# B&R Automation Studio project IntelliRack
Automation Studio 3.0.80.25

## Logical view

Binary libraries used (declarations not repeated): Visapi, runtime, operator, DataObj, Convert, asstring, AsMath, AsIOAcc

### Global.typ
```iecst
TYPE
	color : STRUCT
		fore	:USINT;
		back	:USINT;
	END_STRUCT;
			ctrlPassword : STRUCT
		levelDatapoint	:UINT;
	END_STRUCT;
			ctrlStatusDatapoint : STRUCT
		ctrlHide	:BOOL;
		ctrlLock	:BOOL;
		ctrlFocus	:BOOL;
		ctrlTouchpad	:BOOL;
		statTouchpad	:BOOL;
		statPressLocked	:BOOL;
		statFocus	:BOOL;
		statEdit	:BOOL;
	END_STRUCT;
			greiferParameter : STRUCT
		pulseWidth	:INT;
		periodDuration	:UINT;
		pulseWidthCurrent	:INT;
		periodDurationCurrent	:UINT;
	END_STRUCT;
			tInp : STRUCT
		overloadDC	:BOOL;
		liftHighLim	:BOOL;
		liftLowLim	:BOOL;
		liftPositionClock	:BOOL;
		wireCoilStrtRight	:BOOL;
		wireCoilStrtLeft	:BOOL;
		wireCoilStpRight	:BOOL;
		wireCoilStpLeft	:BOOL;
		wireCoilEmptyRight	:BOOL;
		wireCoilEmptyLeft	:BOOL;
		sthInPos	:BOOL;
		porStopPos	:BOOL;
		clewJam	:BOOL;
		airPresureOk	:BOOL;
		oilLevelLow	:BOOL;
		oilPresureOk	:BOOL;
		zPosStepper	:BOOL;
		supLeftOff	:BOOL;
		supRightOff	:BOOL;
		supLeftOn	:BOOL;
		supRightOn	:BOOL;
		emgCtrl	:BOOL;
		emgBtn	:BOOL;
		strtBtn	:BOOL;
		stpBtn	:BOOL;
		potiClock	:BOOL;
		potiDirection	:BOOL;
		safetySwitch	:BOOL;
		benderNbr1	:BOOL;
		greaseMainGearOk	:BOOL;
		greaseMainGearErr	:BOOL;
		greaseStepWheelOk	:BOOL;
		greaseStepWheelErr	:BOOL;
	END_STRUCT;
			tStepperControl : STRUCT
		switchOn	:BOOL;
		enbleVoltage	:BOOL;
		quickStop	:BOOL;
		enableOperation	:BOOL;
		faultReset	:BOOL;
		rMotorIdent	:BOOL;
		rResetWarning	:BOOL;
	END_STRUCT;
			tStepperIfIn : STRUCT
		absPosActVal	:DINT;
		status	:UINT;
		inputStatus	:USINT;
	END_STRUCT;
			tStepperIfOut : STRUCT
		absPosSetVal	:DINT;
		control	:UINT;
		mode	:SINT;
	END_STRUCT;
			tStepperStatus : STRUCT
		readyToSwitchOn	:BOOL;
		switchedOn	:BOOL;
		operationEnabled	:BOOL;
		fault	:BOOL;
		voltageEnabled	:BOOL;
		quickStop	:BOOL;
		switchOnDisabeld	:BOOL;
		warning	:BOOL;
		targetReached	:BOOL;
	END_STRUCT;
END_TYPE
```

### Global.var
```iecst
VAR
	Inp	:tInp;
	PeriodDurationPWM01PWM02	:UINT;
	PulseWidthCurrentPWM01	:INT;
	TaskNr	:UINT;
	currentPage	:UINT;
	movePointRef	:ARRAY [0..3] OF BOOL;
	moveStepperNegative	:ARRAY [0..3] OF BOOL;
	moveStepperPositive	:ARRAY [0..3] OF BOOL;
	movesteppos	:DINT;
	rPointReached	:BOOL;
	stStepperControl	:ARRAY [0..3] OF tStepperControl;
	stStepperIfIn	:ARRAY [0..3] OF tStepperIfIn;
	stStepperIfOut	:ARRAY [0..3] OF tStepperIfOut;
	stStepperStatus	:ARRAY [0..3] OF tStepperStatus;
END_VAR
```

### Program Logical/test (IEC, version 1.00.0)

#### testCyclic.ab
```automation-basic
PROGRAM _CYCLIC
(* cyclic program *)

loop	idxDrive	:=	1	to	3	do
	if	(moveToPointRef[idxDrive]=TRUE) or (moveToPointRefAll=TRUE) then
		movePointRef[idxDrive]	:=	1
	else
		movePointRef[idxDrive]	:=	0
	endif
endloop
END_PROGRAM
```

#### test.var
```iecst
VAR
	idxDrive	:DINT;
	moveToPointRef	:ARRAY [0..3] OF BOOL;
	moveToPointRefAll	:BOOL;
END_VAR
```

### Program Logical/sthstep (IEC, version 1.02.0)

#### sthstepCyclic.ab
```automation-basic
PROGRAM _CYCLIC
(* cyclic program *)

; V1.00 	sva		2009-06-17	New
; V1.01
; V1.02		sva		2009-08-14	Handling of restart after emergency stop changed

loop idxDrive:= 1 to 3 do

	speedJog[idxDrive]	:= 20*speedJogOptions[idxDrive]

	gearFactor[idxDrive]				:=  (real(driveStepPerRevolution[idxDrive]) * real(microStepPerDriveStep[idxDrive]) * real(gearZ2[idxDrive]) ) / (real(gearZ1[idxDrive]) * real(gearSlope[idxDrive]))
	referencePositionMicroStep[idxDrive]	:= dint(real(referencePositionMM[idxDrive]) * gearFactor[idxDrive])

	; Get status bits
	; ---------------

	stStepperStatus[idxDrive].readyToSwitchOn		:= bit_tst(stStepperIfIn[idxDrive].status, 0)
	stStepperStatus[idxDrive].switchedOn				:= bit_tst(stStepperIfIn[idxDrive].status, 1)
	stStepperStatus[idxDrive].operationEnabled	:= bit_tst(stStepperIfIn[idxDrive].status, 2)
	stStepperStatus[idxDrive].fault							:= bit_tst(stStepperIfIn[idxDrive].status, 3)
	stStepperStatus[idxDrive].voltageEnabled		:= bit_tst(stStepperIfIn[idxDrive].status, 4)
	stStepperStatus[idxDrive].quickStop					:= bit_tst(stStepperIfIn[idxDrive].status, 5)
	stStepperStatus[idxDrive].switchOnDisabeld	:= bit_tst(stStepperIfIn[idxDrive].status, 6)
	stStepperStatus[idxDrive].warning						:= bit_tst(stStepperIfIn[idxDrive].status, 7)
	stStepperStatus[idxDrive].targetReached			:= bit_tst(stStepperIfIn[idxDrive].status, 10)

	; Drive activated and emergency stopp not pressed
	if (driveActive[idxDrive] = 1) then

		; New referencing
		if (referenceSet[idxDrive] = 255) then
			stStepperControl[idxDrive].enbleVoltage			:= 0
			stStepperControl[idxDrive].quickStop				:= 0
			stStepperControl[idxDrive].switchOn					:= 0
			stStepperControl[idxDrive].enableOperation	:= 0
			referenceSet[idxDrive]											:= 0
			sStepper[idxDrive]													:= sTEP_INIT
		endif

		; State machine stepper
		; ---------------------

		; Emergency stop pressed
;		if (Inp.emgCtrl = 1) then
;			sStepper[idxDrive]	:= sTEP_EMERGENCY_STOP
;		endif

		; Stepper error
		if (stStepperStatus[idxDrive].fault = 1) then
			sStepper[idxDrive]	:= sTEP_ERROR
		endif

		case sStepper[idxDrive] of

			action 0:	; Init step

				stStepperControl[idxDrive].enbleVoltage	:= 1
				stStepperControl[idxDrive].quickStop		:= 1

				if (stStepperStatus[idxDrive].readyToSwitchOn = 1) then

					stStepperControl[idxDrive].switchOn	:= 1

					if (stStepperStatus[idxDrive].switchedOn = 1) then

						stStepperControl[idxDrive].enableOperation	:= 1

						; Drive reference not set
						if (referenceSet[idxDrive] = 0) and (referenceUsed[idxDrive]=TRUE) then
							sStepper[idxDrive]						:= sTEP_MOVE_REFERENCE
							stStepperIfOut[idxDrive].mode	:= modeReference[idxDrive]
						endif

						; Drive reference is set
						if (referenceSet[idxDrive] = 1) or (referenceUsed[idxDrive]=FALSE) then
							sStepper[idxDrive]						:= sTEP_WAIT
							stStepperIfOut[idxDrive].mode	:= mODE_MOVE_POSITION
						endif
					endif
				endif

			endaction

			action 12:	; sTEP_MOVE_REFERENCE

				; Refenece sensor reached
				if (stStepperStatus[idxDrive].targetReached = 1) then
					sStepper[idxDrive]										:= sTEP_SET_REFERENCE_POSITION
					stStepperIfOut[idxDrive].absPosSetVal	:= referencePositionMicroStep[idxDrive]
				endif

			endaction

			action 14:	; sTEP_SET_REFERENCE_POSITION

				; Reference position set
				if (stStepperStatus[idxDrive].targetReached = 1) then
					stStepperIfOut[idxDrive].mode	:= mODE_SET_POSITION
					sStepper[idxDrive]						:= sTEP_WAIT
					referenceSet[idxDrive]				:= 1
					firstMovement[idxDrive]				:= 1
					timerStartUp[idxDrive]				:= 0
				endif

			endaction

			action 20:	; sTEP_WAIT

				if (timerStartUp[idxDrive] <= 200) then
					inc(timerStartUp[idxDrive])
				endif

				; Automatic moving
(*				if (movePos[idxDrive] = 1) then
					; Drive stopped
					if (stStepperStatus[idxDrive].targetReached = 1) and (timerStartUp[idxDrive] > 200) then
						if (oldSetPosition[idxDrive] <> setPosition[idxDrive]) or (firstMovement[idxDrive] = 1) then
							firstMovement[idxDrive]		:= 0
							oldSetPosition[idxDrive]	:= setPosition[idxDrive]
							stStepperIfOut[idxDrive].absPosSetVal	:= (dint(   ((setPosition[idxDrive] / 2)+ mOVING_OFFSET) * gearFactor[idxDrive]))
							stStepperIfOut[idxDrive].mode					:= mODE_MOVE_POSITION
							sStepper[idxDrive]										:= sTEP_MOVE_APPROX_POS
							timer[idxDrive]												:= 0
						endif
					endif
				else
*)
					if (moveStepperPositive[idxDrive]=TRUE) and not (endPointPositive[idxDrive] < stStepperIfIn[idxDrive].absPosActVal) then
						stStepperIfOut[idxDrive].absPosSetVal	:= speedJog[idxDrive]
						stStepperIfOut[idxDrive].mode					:= mODE_MOVE_JOG
						sStepper[idxDrive]										:= sTEP_MOVE_JOG
					else if (moveStepperNegative[idxDrive]=TRUE) and not (endPointNegative[idxDrive] > stStepperIfIn[idxDrive].absPosActVal) then
						stStepperIfOut[idxDrive].absPosSetVal	:= -speedJog[idxDrive]
						stStepperIfOut[idxDrive].mode					:= mODE_MOVE_JOG
						sStepper[idxDrive]										:= sTEP_MOVE_JOG
					else if	(setPointZero[idxDrive]=TRUE)	then
						zeroPoint[idxDrive]										:= stStepperIfIn[idxDrive].absPosActVal
						refPointMove[idxDrive]								:= DINT(((REAL(refPoint[idxDrive])+REAL(zeroPoint[idxDrive]))/1024)*200*256)
					else if (movePointRef[idxDrive]=TRUE) then
						stStepperIfOut[idxDrive].absPosSetVal	:= refPointMove[idxDrive]
						stStepperIfOut[idxDrive].mode					:= mODE_MOVE_POSITION
						sStepper[idxDrive]										:= sTEP_MOVE_APPROX_POS
					else if (currentPage = 0) then
						stStepperIfOut[1].absPosSetVal				:= movesteppos
						stStepperIfOut[1].mode								:= mODE_MOVE_POSITION
						sStepper[1]														:= 30
					endif
;				endif

				; Switch on disabled
				if (stStepperStatus[idxDrive].switchOnDisabeld = 1) then
					stStepperControl[idxDrive].switchOn	:= 0
					sStepper[idxDrive]									:= sTEP_SHUTDOWN
				endif

			endaction

			action 21: ;sTEP_MOVE_APPROX_POS

				; Moved to set position + offset
				if (stStepperStatus[idxDrive].targetReached = 1) then
					stStepperIfOut[idxDrive].absPosSetVal	:= refPointMove[idxDrive]
					stStepperIfOut[idxDrive].mode					:= mODE_MOVE_POSITION
					sStepper[idxDrive]										:= sTEP_MOVE_FINE_POS
				endif

				; Switch on disabled
				if (stStepperStatus[idxDrive].switchOnDisabeld = 1) then
					stStepperControl[idxDrive].switchOn	:= 0
					sStepper[idxDrive]									:= sTEP_SHUTDOWN
				endif

			endaction

			action 22:		; sTEP_MOVE_FINE_POS

				; Moved to set position
				if (stStepperStatus[idxDrive].targetReached = 1) then
					sStepper[idxDrive]	:= sTEP_WAIT
				endif

				; Switch on disabled
				if (stStepperStatus[idxDrive].switchOnDisabeld=1) then
					stStepperControl[idxDrive].switchOn	:= 0
					sStepper[idxDrive]									:= sTEP_SHUTDOWN
				endif

			endaction

			action 23: ; sTEP_MOVE_JOG

			endPointNegative[1]	:= zeroPoint[1] - 2200
			endPointNegative[2]	:= zeroPoint[2] - 3800
			endPointNegative[3]	:= zeroPoint[3] - 1280 - 59

			endPointPositive[1]	:= zeroPoint[1] + 2304
			endPointPositive[2]	:= zeroPoint[2]
			endPointPositive[3]	:= zeroPoint[3] - 59

				; Switch on disabled
				if (stStepperStatus[idxDrive].switchOnDisabeld = 1) then
					stStepperControl[idxDrive].switchOn	:= 0
					sStepper[idxDrive]									:= sTEP_SHUTDOWN
				endif

				if ((moveStepperPositive[idxDrive]=FALSE) or (endPointPositive[idxDrive] < stStepperIfIn[idxDrive].absPosActVal)) and ((moveStepperNegative[idxDrive]=FALSE) or (endPointNegative[idxDrive] > stStepperIfIn[idxDrive].absPosActVal)) then
					stStepperIfOut[idxDrive].absPosSetVal	:= 0
					sStepper[idxDrive]										:= sTEP_SHUTDOWN
				endif

			endaction

			action 24:	;sTEP_MOVE_REF

				; Switch on disabled
				if (stStepperStatus[idxDrive].switchOnDisabeld = 1) then
					stStepperControl[idxDrive].switchOn	:= 0
					sStepper[idxDrive]									:= sTEP_SHUTDOWN
				endif

				if (movePointRef[idxDrive]=FALSE) then
					sStepper[idxDrive]	:= sTEP_WAIT
				endif

			endaction

			action 25:	; sTEP_SHUTDOWN

				; Switch on enabled
				if (stStepperStatus[idxDrive].switchOnDisabeld = 0) then
					stStepperControl[idxDrive].switchOn	:= 1
					sStepper[idxDrive]									:= sTEP_WAIT
				endif

			endaction

			action 30:
				if (stStepperStatus[idxDrive].switchOnDisabeld = 1) then
					stStepperControl[idxDrive].switchOn	:= 0
					sStepper[idxDrive]									:= sTEP_SHUTDOWN
				endif

				if 1 = 1 then
					sStepper[idxDrive]	:= sTEP_WAIT
				endif

			endaction

			action 250:	; Emergency stopp

				stStepperControl[idxDrive].enableOperation	:= 0

				; Emergency stop released
				if (Inp.emgCtrl=0) then
					stStepperControl[idxDrive].enbleVoltage	:= 1
					stStepperControl[idxDrive].quickStop		:= 1
					sStepper[idxDrive]											:= sTEP_INIT
				endif

			endaction

			action 255:	; Error step

				stStepperControl[idxDrive].enbleVoltage			:= 0
				stStepperControl[idxDrive].quickStop				:= 0
				stStepperControl[idxDrive].switchOn					:= 0
				stStepperControl[idxDrive].enableOperation	:= 0
				stStepperControl[idxDrive].faultReset				:= 1

				if (stStepperStatus[idxDrive].fault=0) then
					stStepperControl[idxDrive].enbleVoltage	:= 1
					stStepperControl[idxDrive].quickStop		:= 1
					sStepper[idxDrive]											:= sTEP_INIT
				endif

			endaction

		endcase

	; Not active
	else

		stStepperControl[idxDrive].enbleVoltage			:= 0
		stStepperControl[idxDrive].quickStop				:= 0
		stStepperControl[idxDrive].switchOn					:= 0
		stStepperControl[idxDrive].enableOperation	:= 0
		oldWireLengthMM[idxDrive]										:= 0
		sStepper[idxDrive]													:= sTEP_INIT
		referenceSet[idxDrive]											:= 0

	endif

	; Set control word
	; ----------------

	if (stStepperControl[idxDrive].switchOn=1) then
		stStepperIfOut[idxDrive].control	:= bit_set(stStepperIfOut[idxDrive].control, 0)
	else
		stStepperIfOut[idxDrive].control	:= bit_clr(stStepperIfOut[idxDrive].control, 0)
	endif

	if (stStepperControl[idxDrive].enbleVoltage=1) then
		stStepperIfOut[idxDrive].control	:= bit_set(stStepperIfOut[idxDrive].control, 1)
	else
		stStepperIfOut[idxDrive].control	:= bit_clr(stStepperIfOut[idxDrive].control, 1)
	endif

	if (stStepperControl[idxDrive].quickStop=1) then
		stStepperIfOut[idxDrive].control	:= bit_set(stStepperIfOut[idxDrive].control, 2)
	else
		stStepperIfOut[idxDrive].control	:= bit_clr(stStepperIfOut[idxDrive].control, 2)
	endif

	if (stStepperControl[idxDrive].enableOperation=1) then
		stStepperIfOut[idxDrive].control	:= bit_set(stStepperIfOut[idxDrive].control, 3)
	else
		stStepperIfOut[idxDrive].control	:= bit_clr(stStepperIfOut[idxDrive].control, 3)
	endif

	if (stStepperControl[idxDrive].faultReset=1) then
		stStepperControl[idxDrive].faultReset	:= 0
		stStepperIfOut[idxDrive].control				:= bit_set(stStepperIfOut[idxDrive].control, 7)
	else
		stStepperIfOut[idxDrive].control	:= bit_clr(stStepperIfOut[idxDrive].control, 7)
	endif

	if (stStepperControl[idxDrive].rMotorIdent=1) then
		stStepperControl[idxDrive].rMotorIdent	:= 0
		stStepperIfOut[idxDrive].control					:= bit_set(stStepperIfOut[idxDrive].control, 11)
	else
		stStepperIfOut[idxDrive].control	:= bit_clr(stStepperIfOut[idxDrive].control, 11)
	endif

	if (stStepperControl[idxDrive].rResetWarning=1) then
		stStepperControl[idxDrive].rResetWarning	:= 0
		stStepperIfOut[idxDrive].control						:= bit_set(stStepperIfOut[idxDrive].control, 12)
	else
		stStepperIfOut[idxDrive].control	:= bit_clr(stStepperIfOut[idxDrive].control, 12)
	endif

	if (stStepperControl[idxDrive].enableOperation=1) then
		stStepperIfOut[idxDrive].control	:= bit_set(stStepperIfOut[idxDrive].control, 14)
	else
		stStepperIfOut[idxDrive].control	:= bit_clr(stStepperIfOut[idxDrive].control, 14)
	endif

	; MMI aufgestartet d.h. alle Daten aktuell
;	if (dMMI.picture.idxActPic<>0) then
		driveActive[idxDrive]	:= 1
;	endif

endloop
END_PROGRAM
```

#### sthstepInit.ab
```automation-basic
PROGRAM _INIT
(* init program *)
inc(TaskNr)

speedJogOptions[1]	:=	25
speedJogOptions[2]	:=	15
speedJogOptions[3]	:=	10

refPoint[1]	:=	1152
refPoint[2]	:=	-1733
refPoint[3]	:=	-59

zeroPoint[2]	:=	4000

loop idxDrive:= 1 to 3 do

	referenceUsed[idxDrive]	:= FALSE

	sStepper[idxDrive]			:= sTEP_INIT
	referenceSet[idxDrive]	:= 0
	driveActive[idxDrive]		:= 0					; Nicht aktivieren bis alle Daten vorhanden sind
	movePos[idxDrive]				:= 0					; Automatisches Fahren deaktivieren
	modeReference[idxDrive]	:= -128

	; Init control word
	; -----------------

	stStepperControl[idxDrive].switchOn					:= 0
	stStepperControl[idxDrive].enbleVoltage			:= 1
	stStepperControl[idxDrive].quickStop				:= 1
	stStepperControl[idxDrive].enableOperation	:= 0
	stStepperControl[idxDrive].faultReset				:= 0
	stStepperControl[idxDrive].rMotorIdent			:= 0
	stStepperControl[idxDrive].rResetWarning		:= 0

	;========================================
	;	Step Umrechnung
	;========================================

	gearZ1[idxDrive]									:= 15				; Getriebe Zähnezahl Antrieb
	gearZ2[idxDrive]									:= 40				; Getriebe Zähnezahl Abtrieb
	gearSlope[idxDrive]								:= 2.0			; Steigung Gewindestange
	driveStepPerRevolution[idxDrive]	:= 200			; Steps per drive turning
	microStepPerDriveStep[idxDrive] 	:= 256			; Microsteps of X20 stepper module

	referencePositionMM[idxDrive]			:= real(initPosition[idxDrive]) / 1000			; Resulting (wire length / 2) at reference position

	gearFactor[idxDrive]									:=  (real(driveStepPerRevolution[idxDrive]) * real(microStepPerDriveStep[idxDrive]) * real(gearZ2[idxDrive]) ) / (real(gearZ1[idxDrive])* real(gearSlope[idxDrive]))
	referencePositionMicroStep[idxDrive]	:= dint(real(referencePositionMM[idxDrive]) * gearFactor[idxDrive])

endloop
END_PROGRAM
```

#### sthstep.var
```iecst
VAR RETAIN
	initPosition	:ARRAY [0..3] OF UINT;
END_VAR

VAR CONSTANT
	sTEP_INIT	:USINT	:=0;
	sTEP_EMERGENCY_STOP	:UINT	:=250;
	sTEP_ERROR	:USINT	:=255;
	sTEP_MOVE_REFERENCE	:USINT	:=12;
	mODE_MOVE_POSITION	:SINT	:=1;
	sTEP_WAIT	:USINT	:=20;
	sTEP_SET_REFERENCE_POSITION	:USINT	:=14;
	sTEP_SHUTDOWN	:UINT	:=25;
	mOVING_OFFSET	:REAL	:=0.5;
	sTEP_MOVE_APPROX_POS	:USINT	:=21;
	sTEP_MOVE_FINE_POS	:USINT	:=22;
	mODE_SET_POSITION	:SINT	:=-122;
	mODE_MOVE_JOG	:SINT	:=2;
	sTEP_MOVE_JOG	:UINT	:=23;
	sTEP_MOVE_REF	:USINT	:=24;
END_VAR

VAR
	sStepper	:ARRAY [0..3] OF UINT;
	idxDrive	:USINT;
	stStepperStatus	:ARRAY [0..3] OF tStepperStatus;
	stStepperIfIn	:ARRAY [0..3] OF tStepperIfIn;
	stStepperControl	:ARRAY [0..3] OF tStepperControl;
	wireLengthPositionMM	:ARRAY [0..3] OF REAL;
	referenceSet	:ARRAY [0..3] OF USINT;
	modeReference	:ARRAY [0..3] OF SINT;
	timerStartUp	:ARRAY [0..3] OF UDINT;
	gearZ1	:ARRAY [0..3] OF UDINT;
	gearZ2	:ARRAY [0..3] OF UDINT;
	gearSlope	:ARRAY [0..3] OF REAL;
	microStepPerDriveStep	:ARRAY [0..3] OF UINT;
	driveStepPerRevolution	:ARRAY [0..3] OF UDINT;
	gearFactor	:ARRAY [0..3] OF REAL;
	referencePositionMM	:ARRAY [0..3] OF REAL;
	pMMI	:UDINT;
	gPvXGetAdr	:UINT;
	size	:UINT;
	firstMovement	:ARRAY [0..3] OF USINT;
	stStepperIfOut	:ARRAY [0..3] OF tStepperIfOut;
	wireLengthMM	:ARRAY [0..3] OF REAL;
	oldWireLengthMM	:ARRAY [0..3] OF REAL;
	timer	:ARRAY [0..3] OF INT;
	referencePositionMicroStep	:ARRAY [0..3] OF DINT;
	movePos	:ARRAY [0..3] OF USINT;
	wireLengthOffsetMM	:ARRAY [0..3] OF REAL;
	driveActive	:ARRAY [0..3] OF USINT;
	speedJogOptions	:ARRAY [0..3] OF DINT;
	referenceUsed	:ARRAY [0..3] OF BOOL;
	setPosition	:ARRAY [0..3] OF REAL;
	oldSetPosition	:ARRAY [0..3] OF REAL;
	moveStepperPositive	:ARRAY [0..3] OF BOOL;
	speedJog	:ARRAY [0..3] OF DINT;
	moveStepperNegative	:ARRAY [0..3] OF BOOL;
	moveStepperReference	:ARRAY [0..3] OF BOOL;
	refPoint	:ARRAY [0..3] OF DINT;
	setPointZero	:ARRAY [0..3] OF BOOL;
	zeroPoint	:ARRAY [0..3] OF DINT;
	refPointMove	:ARRAY [0..3] OF DINT;
	detail1	:USINT;
	detail2	:USINT;
	detail4	:USINT;
	detail3	:USINT;
	endPointPositive	:ARRAY [0..3] OF DINT;
	endPointNegative	:ARRAY [0..3] OF DINT;
END_VAR
```

### Program Logical/greifer (IEC, version 1.00.0)

#### greiferCyclic.ab
```automation-basic
PROGRAM _CYCLIC
(* cyclic program *)

if (moveGreiferPositive=TRUE) then
	greifer.pulseWidthCurrent			:=	greifer.pulseWidth
	greifer.periodDurationCurrent	:=	greifer.periodDuration
else if (moveGreiferNegative=TRUE) then
	greifer.pulseWidthCurrent			:=	-greifer.pulseWidth
	greifer.periodDurationCurrent	:=	greifer.periodDuration
else
	greifer.pulseWidthCurrent			:=	0
	greifer.periodDurationCurrent	:=	0
endif
END_PROGRAM
```

#### greiferInit.ab
```automation-basic
PROGRAM _INIT
(* init program *)

;Frequenz							us pro Zyklus
greifer.pulseWidth			:=	5000

;Anteil in "Prozent" (UINT) von 1/-1 Signal
greifer.periodDuration	:=	20
END_PROGRAM
```

#### greifer.var
```iecst
VAR
	moveGreiferPositive	:BOOL;
	moveGreiferNegative	:BOOL;
	greifer	:greiferParameter;
END_VAR
```

### Program Logical/ctrlvisu (IEC, version 0.00.0)

#### ctrlvisuCyclic.ab
```automation-basic
PROGRAM _CYCLIC
(* cyclic program *)

if detail1 = 0 then
	detail1focus := 2
else if detail2 = 0 then
	detail1focus := 2
else if detail3 = 0 then
	detail1focus := 2
else if detail4 = 0 then
	detail1focus := 2
else
	detail1focus := 0
	detail2focus := 0
	detail3focus := 0
	detail4focus := 0
endif

if ready <> 1 then
	VC_HANDLE = VA_Setup(1, "visu")

	if	VC_HANDLE <> 0 then
		ready = 1
	endif
endif

loop idx :=	1 to 5 do

	statusDatapoint[idx].statTouchpad			:=	bit_tst(ctrlWord[idx], 12)
	statusDatapoint[idx].statPressLocked	:=	bit_tst(ctrlWord[idx], 13)
	statusDatapoint[idx].statFocus				:=	bit_tst(ctrlWord[idx], 14)
	statusDatapoint[idx].statEdit					:=	bit_tst(ctrlWord[idx], 15)

endloop
if currentPage <> 0 then
	CASE	achsenwahl of
		action 1:
			if statusDatapoint[5].statFocus = 0 then
				statusDatapoint[1].ctrlHide = 1

				achsenwahl :=	2
			endif
		endaction

		action 2:

			if VA_Saccess(1, VC_HANDLE)= 0 then

				VA_GetTouchAction(1, VC_HANDLE, 0, UDINT(ADR(touch2)))

				if (touch2.status = 1) and (touch2.x > 255) and (touch2.x < 385) and (touch2.y > 420) and (detail1 = 1) and (detail2 = 1) and (detail3 = 1) and (detail4 = 1)then
					statusDatapoint[1].ctrlHide = 0

					achsenwahl := 3
				endif

				VA_Srelease(1, VC_HANDLE)
			endif
		endaction

		action 3:

			if ready = 1 then
				if VA_Saccess(1, VC_HANDLE)= 0 then

					VA_GetTouchAction(1, VC_HANDLE, 0, UDINT(ADR(touch2)))

					if touch2.status = 1 then
						if (touch2.x > 255) and (touch2.x < 385) and (touch2.y > 420) then
							idxbmp	:=	0
						else if (touch2.x > 255) and (touch2.x < 385) and (touch2.y > 380) then
							idxbmp	:=	1
						else if (touch2.x > 255) and (touch2.x < 385) and (touch2.y > 340) then
							idxbmp	:=	2
						else if (touch2.x > 255) and (touch2.x < 385) and (touch2.y > 300) then
							idxbmp	:=	3
						else if (touch2.x > 255) and (touch2.x < 385) and (touch2.y > 260) then
							idxbmp	:=	4
						else
							idxbmp	:=	0
						endif
					else if touch2.status = 2 then
						if (touch2.x > 255) and (touch2.x < 385) and (touch2.y > 420) then
							changePage	:=	12
							achsenwahl	:=	1
						else if (touch2.x > 255) and (touch2.x < 385) and (touch2.y > 380) then
							changePage	:=	6
							achsenwahl	:=	1
						else if (touch2.x > 255) and (touch2.x < 385) and (touch2.y > 340) then
							changePage	:=	7
							achsenwahl	:=	1
						else if (touch2.x > 255) and (touch2.x < 385) and (touch2.y > 300) then
							changePage	:=	3
							achsenwahl	:=	1
						else if (touch2.x > 255) and (touch2.x < 385) and (touch2.y > 260) then
							changePage	:=	4
							achsenwahl	:=	1
						endif
					endif

					VA_Srelease(1, VC_HANDLE)

				endif
			endif
		endaction
	endcase
endif

loop idx := 1 to 5 do

	if statusDatapoint[idx].ctrlFocus = 1 then
		ctrlWord[idx]	:=	bit_set(ctrlWord[idx], 3)
	else if statusDatapoint[idx].ctrlFocus = 0 then
		ctrlWord[idx]	:=	bit_clr(ctrlWord[idx], 3)
	endif

	if statusDatapoint[idx].ctrlLock = 1 then
		ctrlWord[idx]	:=	bit_set(ctrlWord[idx], 1)
	else if statusDatapoint[idx].ctrlLock = 0 then
		ctrlWord[idx]	:=	bit_clr(ctrlWord[idx], 1)
	endif

	if statusDatapoint[idx].ctrlHide = 1 then
		ctrlWord[idx]	:=	bit_set(ctrlWord[idx], 0)
	else if statusDatapoint[idx].ctrlHide = 0 then
		ctrlWord[idx]	:=	bit_clr(ctrlWord[idx], 0)
	endif

	if statusDatapoint[idx].ctrlTouchpad = 1 then
		ctrlWord[idx]	:=	bit_set(ctrlWord[idx], 2)
	else if statusDatapoint[idx].ctrlTouchpad = 0 then
		ctrlWord[idx]	:=	bit_clr(ctrlWord[idx], 2)
	endif
endloop

;Damit die Visualisierung da Passwort ausführen kann
password.levelDatapoint
END_PROGRAM
```

#### ctrlvisuInit.ab
```automation-basic
PROGRAM _INIT
(* init program *)

achsenwahl := 1

detail1 := 1
detail2 := 1
detail3 := 1
detail4 := 1

detail1focus := 0
detail2focus := 0
detail3focus := 0
detail4focus := 0
END_PROGRAM
```

#### ctrlvisu.var
```iecst
VAR
	statusDatapoint	:ARRAY [0..5] OF ctrlStatusDatapoint;
	ctrlWord	:ARRAY [0..5] OF UINT;
	lock	:BOOL;
	hide	:BOOL;
	touchpad	:BOOL;
	focus	:BOOL;
	idx	:UINT;
	achsenwahl	:UINT;
	ready	:BOOL;
	VC_HANDLE	:UDINT;
	test	:BOOL;
	touch2	:TouchAction;
	changePage	:UINT;
	idxbmp	:UINT;
	password	:ctrlPassword;
	durchgang1	:BOOL;
	detail4	:UINT;
	detail1	:UINT;
	detail2	:UINT;
	detail3	:UINT;
	detail1focus	:UINT;
	detail2focus	:UINT;
	detail3focus	:UINT;
	detail4focus	:UINT;
END_VAR
```

### Program Logical/stepmove (IEC, version 0.00.0)

#### stepmoveCyclic.ab
```automation-basic
PROGRAM _CYCLIC
(* cyclic program *)

;Wenn die aktuelle Seite die Experimentierseite ist
if currentPage = 0 then

	;Bildschirm bereit zum Bearbeiten
	if ready <> 1 then
		VC_HANDLE = VA_Setup(1, "visu")

		if	VC_HANDLE <> 0 then
			ready = 1
		endif
	endif

	;Wenn Bildschirm bereit zum Bearbeiten
	if ready = 1 then

		;Erster Durchlauf Formen zeichnen
		if test = 0 then
			if VA_Saccess(1, VC_HANDLE)= 0 then

				;Mittelpunkt zeichnen
				VA_Rect(1, VC_HANDLE, 239, 239, 3, 3, fill, color)

				;Aktuelle-Position Form zeichnen
				VA_Rect(1, VC_HANDLE, UINT(position_x), UINT(position_y), width, heigth, fill, color)
				test = 1

				VA_Srelease(1, VC_HANDLE)

			endif
		endif

		;Weitere Durchläufe
		if test = 1 then

			if VA_Saccess(1, VC_HANDLE) = 0 then

				;Welche Taste ist aktuell betätigt
				if fest = 1 then
					bewegen = 0
				else if locker = 1 then
					bewegen = 1
					zeichnen = 1
					VA_Redraw(1, VC_HANDLE)
					VA_Rect(1, VC_HANDLE, 239, 239, 3, 3, fill, color)
					VA_Rect(1, VC_HANDLE, UINT(position_x), UINT(position_y), width, heigth, fill, color)
				endif

				;Abfragen der aktuelle Touch-Position
				VA_GetTouchAction(1, VC_HANDLE, 0, UDINT(adr(touch)))

				;Übergabe der Touch-Position Informationen
				x_position = touch.x
				y_position = touch.y
				touch_status = touch.status

				;Wenn Touchpanel betätigt und bewegen erlaubt
				if touch_status = 1 and bewegen = 1 then

					;Abfrage ob Form gegriffen wurde
					if ((x_position) > position_x) and ((x_position) < (position_x + width)) and ((y_position) > position_y) and ((y_position) < (position_y + heigth)) and (packen_erlaubt = 0) and bewegen = 1 then
						packen_erlaubt = 1
						gepackt_x = x_position - position_x
						gepackt_y = y_position - position_y

						;Überschreiben der Drawbox mit weiss
						VA_Rect(1, VC_HANDLE, 0, 0, 480, 480, 15, 15)

						;Mittelpunkt zeichnen
						VA_Rect(1, VC_HANDLE, 239, 239, 3, 3, fill, color)
					endif

					;Wenn Form gegriffen wurde
					if packen_erlaubt = 1 then

						;Letzte Position der Form löschen
						VA_Rect(1, VC_HANDLE, UINT(position_x), UINT(position_y), width, heigth, 15, 15)

						;Mittelpunkt zeichnen
						VA_Rect(1, VC_HANDLE, 239, 239, 3, 3, fill, color)

						;Berechnen der Form-Position
						x1 = x1 + (x_position - x_position_old)
						y1 = y1 + (y_position - y_position_old)

						position_x = x1 - gepackt_x
						position_y = y1 - gepackt_y

						;Berechnen der Richtung und Schritte für Drehtisch
						x_position_EXP	:=	(EXPT(-240+x_position,2))
						y_position_EXP	:=	(EXPT(-240+y_position,2))
						sqrtergebnis		:=	SQRT(EXPT(-240+x_position,2))/SQRT((y_position_EXP)+(x_position_EXP))

						if (x_position < 240) and (y_position < 240) then
							asdasd					:=	ASIN(sqrtergebnis)
							asd							:=	90
						else if (x_position > 240) and (y_position < 240) then
							asdasd					:=	ACOS(sqrtergebnis)
							asd							:=	0
						else if (x_position > 240) and (y_position > 240) then
							asdasd					:=	ASIN(sqrtergebnis)
							asd							:=	-90
						else if (x_position < 240) and (y_position > 240) then
							asdasd					:=	ACOS(sqrtergebnis)
							asd							:=	-180
						endif

						dasdas 					:= (25600*((360*asdasd/amTWOPI)+asd))/360
						dasdasdasdasda	:=	DINT(dasdas)

						movesteppos			:= 9*dasdasdasdasda

						;Drawbox-Begrenzungen
						if ((x_position - gepackt_x + width) > x_stop) then
							position_x = x_stop - width
						else if ((x_position - gepackt_x) < x_start) then
							position_x = x_start
						endif

						if ((y_position - gepackt_y + heigth) > y_stop) then
							position_y = y_stop - heigth
						else if ((y_position - gepackt_y) < y_start) then
							position_y = y_start
						endif

						;Zeichnen der Form
						VA_Rect(1, VC_HANDLE, UINT(position_x), UINT(position_y), width, heigth, fill, color)

						;Speichern der letztn Position
						x_position_old = x_position
						y_position_old = y_position

					endif

				else
					if packen_erlaubt = 1 then
						packen_erlaubt = 0
					endif
				endif

				VA_Srelease(1, VC_HANDLE)
			endif
		endif
	endif
endif
END_PROGRAM
```

#### stepmoveInit.ab
```automation-basic
PROGRAM _INIT
(* init program *)

test 						:= 0
x1 							:= 400
y1 							:= 235
x_position_old 	:= x1
y_position_old 	:= y1

;Startposition der From
position_x 			:= 400
position_y 			:= 235

;Parameter für Begrenzungen vom Zeichen
x_start 				:= 0
x_stop					:= 480
y_start					:= 0
y_stop					:= 480

;Paramter für Form der aktuellen Position
heigth					:=	20
width						:=	20
fill						:=	0
color						:=	0
END_PROGRAM
```

#### stepmove.var
```iecst
VAR
	test	:BOOL;
	ready	:BOOL;
	VC_HANDLE	:UDINT;
	redesign	:BOOL;
	packen_erlaubt	:BOOL;
	fest	:BOOL;
	width	:UINT;
	heigth	:UINT;
	touch_status	:UDINT;
	dasdas	:REAL;
	y_start	:DINT;
	x_start	:DINT;
	fill	:UINT;
	x_position	:DINT;
	zeichnen	:BOOL;
	locker	:BOOL;
	x_position_old	:DINT;
	position_x	:DINT;
	y_position_old	:DINT;
	position_y	:DINT;
	y_position	:DINT;
	touch	:TouchAction;
	y_stop	:DINT;
	x_stop	:DINT;
	bewegen	:BOOL;
	asdasd	:REAL;
	y1	:DINT;
	x1	:DINT;
	color	:UINT;
	gepackt_x	:DINT;
	gepackt_y	:DINT;
	dasdasdasdasda	:DINT;
	x_position_EXP	:REAL;
	y_position_EXP	:REAL;
	sqrtergebnis	:REAL;
	asd	:REAL;
	das	:DINT;
END_VAR
```

### Program Logical/testvisu (IEC, version 0.00.0)

#### testvisuCyclic.ab
```automation-basic
PROGRAM _CYCLIC
(* cyclic program *)

;loop	idx	:=	1	to	8	do
;	color	access	adr	(idxColor[idx])
;	color.fore	:=	100
;	color.back	:=	0
;endloop

if (ready <> 1) then
	VC_HANDLE = VA_Setup(1, "visu")

	if	VC_HANDLE <> 0 then
		ready := 1
	endif
endif

if (ready = 1) and (first = 0) then
	if VA_Saccess(1, VC_HANDLE)= 0 then

		VA_Redraw(1, VC_HANDLE)

		VA_Rect(1, VC_HANDLE, 0, 400, 640, 80, 100, 100)

		VA_Srelease(1, VC_HANDLE)

		first	:=	1

	endif
endif

if (ready = 1) and (first = 1) then
	if VA_Saccess(1, VC_HANDLE)= 0 then

		VA_GetTouchAction(1, VC_HANDLE, 0, UDINT(ADR(touch2)))

			Aktion	:=	BOOL(touch2.status - 1)
			;if touch2.status = 1 then

			if EDGE(Aktion) then
				VA_Rect(1, VC_HANDLE, 0, 320, 640, 80, 15, 15)
			endif

			VA_Rect(1, VC_HANDLE, (80 * (changed - 1)), 400, 80, 80, 100, 100)

			loop	idx:=	1	to	8 do

				if (touch2.x	< (80 * idx)) and (touch2.x > (80 * (idx - 1))) and (touch2.y > 399) then
					if (touch2.status = 1) and (counter2 <> 2) then
						changed	:=	idx
						VA_Rect(1, VC_HANDLE, (80 * (idx - 1)), 400, 80, 80, 10, 10)
						counter := 0
						inc(counter2)
					else if (touch2.status = 2) and (counter <> 2) then
						VA_Rect(1, VC_HANDLE, 0, 320, 640, 80, 15, 15)
						VA_Rect(1, VC_HANDLE, (80 * (idx - 1)), 320, 80, 80, 10, 10)
						counter2 :=	0
						inc(counter)
					endif
				endif

			endloop
			;endif

		VA_Srelease(1, VC_HANDLE)

	endif
endif
END_PROGRAM
```

#### testvisuInit.ab
```automation-basic
PROGRAM _INIT
(* init program *)

first := 0
END_PROGRAM
```

#### testvisu.var
```iecst
VAR
	idx	:UINT;
	ready	:BOOL;
	VC_HANDLE	:UDINT;
	touch2	:TouchAction;
	changed	:UINT;
	first	:BOOL;
	Aktion	:BOOL;
	counter2	:USINT;
	counter	:USINT;
END_VAR
```

### Program Logical/testvisa (IEC, version 0.00.0)

#### testvisaCyclic.ab
```automation-basic
PROGRAM _CYCLIC
(* cyclic program *)

(* cyclic program *)

if (ready <> 1) then
	VC_HANDLE = VA_Setup(1, "visu")

	if	VC_HANDLE <> 0 then
		ready := 1
		if VA_Saccess(1, VC_HANDLE)= 0 then
			VA_Redraw(1, VC_HANDLE)
			VA_Srelease(1, VC_HANDLE)
		endif
	endif
endif

if (ready = 1) then
	if VA_Saccess(1, VC_HANDLE)= 0 then

		VA_Rect(1, VC_HANDLE, UINT(touch2.x-40), UINT(touch2.y-40), 80, 80, 15, 15)

		VA_GetTouchAction(1, VC_HANDLE, 0, UDINT(ADR(touch2)))

		VA_Rect(1, VC_HANDLE, UINT(touch2.x-40), UINT(touch2.y-40), 80, 80, UINT((touch2.x/6.4) + (touch2.y/4.8)), UINT((touch2.x/6.4) + (touch2.y/4.8)))

		VA_Srelease(1, VC_HANDLE)

	endif
endif
END_PROGRAM
```

#### testvisa.var
```iecst
VAR
	ready	:BOOL;
	VC_HANDLE	:UDINT;
	touch2	:TouchAction;
END_VAR
```

### Program Logical/a_soption (IEC, version 0.00.0)

#### a_soptionCyclic.ab
```automation-basic
PROGRAM _CYCLIC
(* cyclic program *)

AsIOAccWrite(1, UDINT(ADR("SL1.SS1.IF2.ST16.IF1.ST3")), UDINT(ADR("ConfigOutput03a")), valueHaltestrom[1], status)
AsIOAccWrite(1, UDINT(ADR("SL1.SS1.IF2.ST16.IF1.ST3")), UDINT(ADR("ConfigOutput04a")), valueNennstrom[1], status)
AsIOAccWrite(1, UDINT(ADR("SL1.SS1.IF2.ST16.IF1.ST3")), UDINT(ADR("ConfigOutput05a")), valueMaximalstrom[1], status)

AsIOAccWrite(1, UDINT(ADR("SL1.SS1.IF2.ST16.IF1.ST6")), UDINT(ADR("ConfigOutput03")), valueHaltestrom[2], status)
AsIOAccWrite(1, UDINT(ADR("SL1.SS1.IF2.ST16.IF1.ST6")), UDINT(ADR("ConfigOutput04")), valueNennstrom[2], status)
AsIOAccWrite(1, UDINT(ADR("SL1.SS1.IF2.ST16.IF1.ST6")), UDINT(ADR("ConfigOutput05")), valueMaximalstrom[2], status)

AsIOAccWrite(1, UDINT(ADR("SL1.SS1.IF2.ST16.IF1.ST6")), UDINT(ADR("ConfigOutput06")), valueHaltestrom[3], status)
AsIOAccWrite(1, UDINT(ADR("SL1.SS1.IF2.ST16.IF1.ST6")), UDINT(ADR("ConfigOutput07")), valueNennstrom[3], status)
AsIOAccWrite(1, UDINT(ADR("SL1.SS1.IF2.ST16.IF1.ST6")), UDINT(ADR("ConfigOutput08")), valueMaximalstrom[3], status)

AsIOAccWrite(1, UDINT(ADR("SL1.SS1.IF2.ST16.IF1.ST3")), UDINT(ADR("MaxAcc01")), (valueAcc[1]*5), status)
AsIOAccWrite(1, UDINT(ADR("SL1.SS1.IF2.ST16.IF1.ST3")), UDINT(ADR("MaxDec01")), (valueDec[1]*5), status)

AsIOAccWrite(1, UDINT(ADR("SL1.SS1.IF2.ST16.IF1.ST3")), UDINT(ADR("MaxSpeed01pos")), (valueMaxSpeed), status)

AsIOAccRead(1, UDINT(ADR("SL1.SS1.IF2.ST16.IF1.ST3")), UDINT(ADR("AbsPos1ActValAcyclic")), status, valueasyncpos)

;AsIOAccWrite(1, UDINT(ADR("SL1.SS1.IF2.ST16.IF1.ST6")), UDINT(ADR("ConfigOutput08")), valueMaximalstrom[3], status)
;AsIOAccWrite(1, UDINT(ADR("SL1.SS1.IF2.ST16.IF1.ST6")), UDINT(ADR("ConfigOutput08")), valueMaximalstrom[3], status)

;AsIOAccWrite(1, UDINT(ADR("SL1.SS1.IF2.ST16.IF1.ST6")), UDINT(ADR("ConfigOutput08")), valueMaximalstrom[3], status)
;AsIOAccWrite(1, UDINT(ADR("SL1.SS1.IF2.ST16.IF1.ST6")), UDINT(ADR("ConfigOutput08")), valueMaximalstrom[3], status)
END_PROGRAM
```

#### a_soptionInit.ab
```automation-basic
PROGRAM _INIT
(* init program *)

;Prozent von 3A

valueHaltestrom[1] 		:= 70
valueNennstrom[1]			:= 90
valueMaximalstrom[1]	:= 100

;Prozent von 6A
valueHaltestrom[2]		:= 50
valueNennstrom[2]			:= 50
valueMaximalstrom[2]	:= 50

valueHaltestrom[3]		:= 50
valueNennstrom[3]			:= 50
valueMaximalstrom[3]	:= 50

;Beschleunigung
valueAcc[1]						:= 3
valueAcc[2]						:= 1
valueAcc[3]						:= 1

;Bremsen
valueDec[1]						:= 3
valueDec[2]						:= 1
valueDec[3]						:= 1

valueMaxSpeed					:= 700
END_PROGRAM
```

#### a_soption.var
```iecst
VAR
	AsIOAccWrite_0	:AsIOAccWrite;
	valueHaltestrom	:ARRAY [0..3] OF UDINT;
	status	:UINT;
	SL1	:UDINT;
	valueNennstrom	:ARRAY [0..3] OF UDINT;
	valueMaximalstrom	:ARRAY [0..3] OF UDINT;
	valueAcc	:ARRAY [0..3] OF UINT;
	valueDec	:ARRAY [0..3] OF UINT;
	valueMaxSpeed	:UINT;
	DatObjRead_0	:DatObjRead;
	valueasyncpos	:UDINT;
	DatObjRead_1	:DatObjRead;
	AsIOAccRead_0	:AsIOAccRead;
END_VAR
```

### Program Logical/sthver (ANSIC, version 0.00.0) - Ermitteln der Softwareversion aus xy.pgp

#### sthver.c
```c
#ifdef _DEFAULT_INCLUDES
 #include <AsDefault.h>
#endif
/********************************
       I N C L U D E
********************************/
#include <bur\plc.h>
#include <bur\plctypes.h>
#include <asstring.h>

#if _OLD_DECLARATION	/* due to conversion */
_LOCAL char szVersion[80];
#endif	/* "#endif" due to conversion */

void _INIT init_sthver(void) {
	char *pszFilename = __FILE__; /* diese Konstante enthält den Filenamen inclusive alle Unterverzeichnisse */
	short i=0;
	short PosChar=0, VerChar=0;

	/* Länge des Filenamens bestimmen */
	while(pszFilename[i]) i++;

	/* Den Filenamen von hinten beginnend nach .pgp absuchen und die Position merken */
	i=i-3;
	while(i>0){
		if( (pszFilename[i]=='.')&&(pszFilename[i+1]=='p')&&(pszFilename[i+2]=='g')&&(pszFilename[i+3]=='p') ){
			PosChar = i;
			break;
		}
		i--;
	}

	/* Anzahl Zeichen bis ersten Backslash vor ".pgp" bestimmen */
	if (PosChar > 0) {
		while (PosChar > VerChar) {
			if (pszFilename[PosChar - VerChar] != '\\' ) VerChar++;
			else {VerChar--; break;}
		}
	}

	/*Version kopieren*/
	memcpy(&szVersion, &pszFilename[PosChar - VerChar], VerChar);
}

void _CYCLIC cyclic_sthver(void) {
/*no code*/
}
```

#### sthver.var
```iecst
VAR
	szVersion	:ARRAY [0..79] OF SINT;
END_VAR
```

- Visualisation Logical/visu (not shown)

Listed in the project but not available here: Logical/test/testInit.ab, Logical/testvisa/testvisaInit.ab
